{attribute 'linkalways'}
{attribute 'hide_all_locals'}
FUNCTION_BLOCK ValueWordRead EXTENDS ValueBase IMPLEMENTS ValueRead
VAR
	thisValue : WORD;
END_VAR

{attribute 'call_after_global_init_slot' := '1'}
{attribute 'call_after_online_change_slot' := '1'}
METHOD PROTECTED GetThisAnyType
VAR_INPUT
END_VAR
thisAnyType := ToAnyType(thisValue);
END_METHOD

METHOD GetAsType : BOOL
VAR_INPUT
	destination : __SYSTEM.AnyType;
END_VAR
GetAsType := ConvertAnyType(thisAnyType, destination);
END_METHOD

METHOD GetAsString : T_MaxString
VAR_INPUT
END_VAR
GetAsString := TO_STRING(thisValue);
END_METHOD

METHOD Get : BOOL
VAR_INPUT
	destination : ANY;
END_VAR
Get := ConvertAnyType(thisAnyType, destination);
END_METHOD

METHOD FB_init : BOOL
VAR_INPUT
	bInitRetains : BOOL; // if TRUE, the retain variables are initialized (warm start / cold start)
	bInCopyCode : BOOL;  // if TRUE, the instance afterwards gets moved into the copy code (online change)
END_VAR
_ValueType := __SYSTEM.TYPE_CLASS.TYPE_WORD;
END_METHOD

{attribute 'monitoring' := 'call'}
PROPERTY Value : WORD
GET
Value := thisValue;
END_GET
END_PROPERTY

END_FUNCTION_BLOCK

(* stored: Version 1.1.0.1
   POU ValueWordRead: Id {cdfdf7e7-1c45-40a9-9d0a-ee842c78b160}, SpecialFunc None
   Method GetThisAnyType: Id {d3e62816-8354-4a8c-8dc0-e037f6f23110}
   Method GetAsType: Id {9191455d-7c97-49a9-bd08-0338b07a323e}
   Method GetAsString: Id {d219ac8c-990a-4414-b1b3-d52397826a25}
   Method Get: Id {cbb28641-3c7a-4515-bae4-e75ff99281c2}
   Method FB_init: Id {5ee01bd0-6510-4f61-b683-f03db934dd21}
   Property Value: Id {c00bf5cc-16b8-4afb-bcff-189aa3014262}
   Get Get: Id {892b4770-6f6a-420b-9d39-375289a0eb6b} *)
